{attribute 'qualified_only'}
{attribute 'strict'}
{attribute 'to_string'}
TYPE AxisDirection :
(
	PositiveDirection,
	NegativeDirection
);
END_TYPE

(* stored: Version 1.1.0.1, ProductVersion 3.1.4026.18
   DUT AxisDirection: Id {1825dbeb-b9cd-0841-3c60-a91072da252a} *)
